# EPICS substitutions: tizrSup/tizr_error_setter.substitutions
file $(UTILITIES)/db/error_setter.template {
    pattern {P, STREAM_PV, PV_NAME}

    {"\$(P)", "\$(P)OUT_OF_RANGE", "DENSITY"}
    {"\$(P)", "\$(P)OUT_OF_RANGE", "TEMPERATURE"}
    {"\$(P)", "\$(P)OUT_OF_RANGE", "CONDITION"}
}
